TYPE CamIn_Statuses_typ :
	STRUCT
		InSync 			: 		BOOL;
		Busy 			: 		BOOL; 
		Active 			: 		BOOL; 
		CommandAborted 	: 		BOOL;

	END_STRUCT
END_TYPE

(* stored: Version 1.1.0.1, ProductVersion 3.1.4024.3
   DUT CamIn_Statuses_typ: Id {a8671b1b-0026-06d6-3607-79b45a4e5dc7} *)
